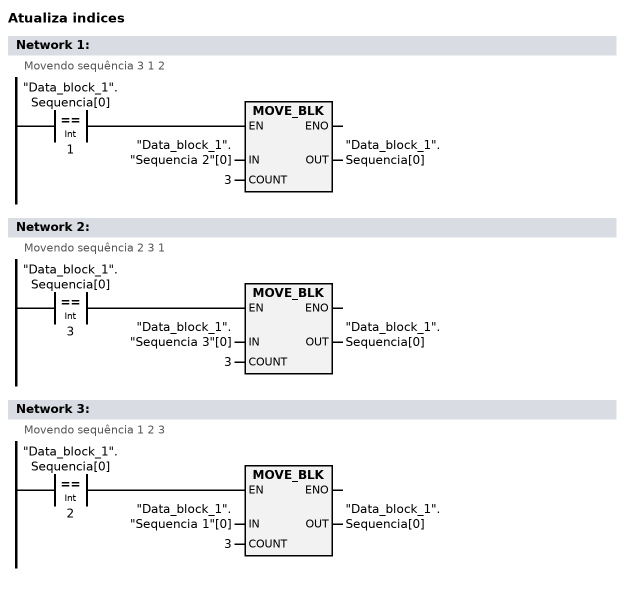
   IF "Data_block_1".Sequencia[0] = 1 THEN
       MOVE_BLK(IN := "Data_block_1"."Sequencia 2"[0], COUNT := 3, OUT => "Data_block_1".Sequencia[0]);
   END_IF;
END_REGION

REGION Network 2
   // Movendo sequência 2 3 1
   IF "Data_block_1".Sequencia[0] = 3 THEN
       MOVE_BLK(IN := "Data_block_1"."Sequencia 3"[0], COUNT := 3, OUT => "Data_block_1".Sequencia[0]);
   END_IF;
END_REGION

REGION Network 3
   // Movendo sequência 1 2 3
   IF "Data_block_1".Sequencia[0] = 2 THEN
       MOVE_BLK(IN := "Data_block_1"."Sequencia 1"[0], COUNT := 3, OUT => "Data_block_1".Sequencia[0]);
   END_IF;
END_REGION
END_FUNCTION

FUNCTION "Relaciona indices" : Void   // FC25, LAD
{ S7_Optimized_Access := 'TRUE' }
VERSION : 0.1
   VAR_INPUT
      index : Int;   // Índice da sequência de compressores
      "valor logico" : Bool;   // Valor que determina se é preciso ligar ou desligar
   END_VAR
   VAR_TEMP   // added for the SCL form of the ladder/FBD networks
      _w1 : Bool;
   END_VAR
BEGIN

REGION Network 1
   // Seta ou reseta caso Sequencia[index] == 1
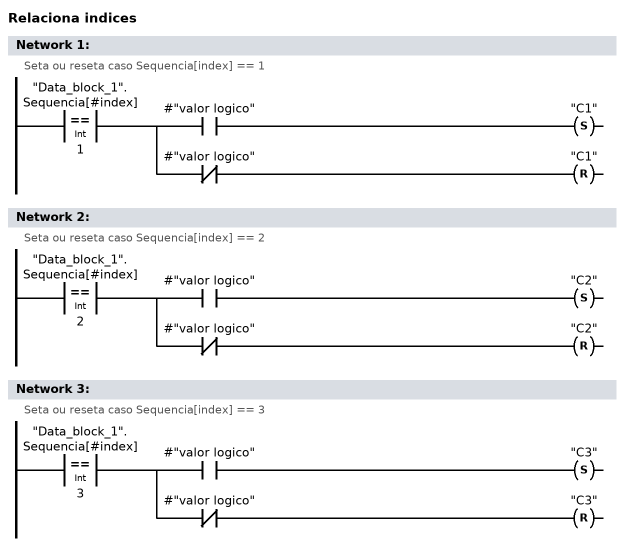
   RUNG wire#powerrail
      { S7_Templates := "SrcType := Int" } EQ_Contact(in1 := "Data_block_1".Sequencia[#index], in2 := 1)
      wire#w1
      Contact( #"valor logico" )
      S_Coil( "C1" )
   END_RUNG
   RUNG wire#w1
      I_Contact( #"valor logico" )
      R_Coil( "C1" )
   END_RUNG
   // the same network as SCL:
   #_w1 := "Data_block_1".Sequencia[#index] = 1;
   IF #_w1 AND #"valor logico" THEN "C1" := TRUE; END_IF;
   IF #_w1 AND NOT #"valor logico" THEN "C1" := FALSE; END_IF;
END_REGION

REGION Network 2
   // Seta ou reseta caso Sequencia[index] == 2
   RUNG wire#powerrail
      { S7_Templates := "SrcType := Int" } EQ_Contact(in1 := "Data_block_1".Sequencia[#index], in2 := 2)
      wire#w1
      Contact( #"valor logico" )
      S_Coil( "C2" )
   END_RUNG
   RUNG wire#w1
      I_Contact( #"valor logico" )
      R_Coil( "C2" )
   END_RUNG
   // the same network as SCL:
   #_w1 := "Data_block_1".Sequencia[#index] = 2;
   IF #_w1 AND #"valor logico" THEN "C2" := TRUE; END_IF;
   IF #_w1 AND NOT #"valor logico" THEN "C2" := FALSE; END_IF;
END_REGION

REGION Network 3
   // Seta ou reseta caso Sequencia[index] == 3
   RUNG wire#powerrail
      { S7_Templates := "SrcType := Int" } EQ_Contact(in1 := "Data_block_1".Sequencia[#index], in2 := 3)
      wire#w1
      Contact( #"valor logico" )
      S_Coil( "C3" )
   END_RUNG
   RUNG wire#w1
      I_Contact( #"valor logico" )
      R_Coil( "C3" )
   END_RUNG
   // the same network as SCL:
   #_w1 := "Data_block_1".Sequencia[#index] = 3;
   IF #_w1 AND #"valor logico" THEN "C3" := TRUE; END_IF;
   IF #_w1 AND NOT #"valor logico" THEN "C3" := FALSE; END_IF;
END_REGION
END_FUNCTION

FUNCTION "M1 - Operacao finalizada" : Void   // FC26, LAD
{ S7_Optimized_Access := 'TRUE' }
VERSION : 0.1
   VAR_TEMP   // added for the SCL form of the ladder/FBD networks
      _w1 : Bool;
   END_VAR
BEGIN

REGION Network 1
   // MODO AUTOMÁTICO [M1] - Operação finalizada
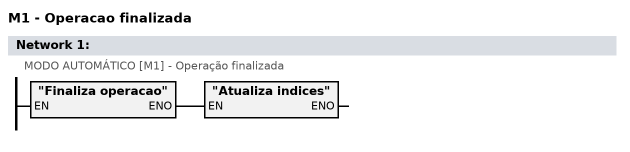
   RUNG wire#powerrail
      "Finaliza operacao"()
      "Atualiza indices"()
   END_RUNG
   // the same network as SCL:
   "Finaliza operacao"(ENO => #_w1);
   IF #_w1 THEN "Atualiza indices"(); END_IF;
END_REGION
END_FUNCTION

FUNCTION "Monitora pressao" : Void   // FC27, LAD
{ S7_Optimized_Access := 'TRUE' }
VERSION : 0.1
   VAR_OUTPUT
      Crescente : Bool;   // Pressão crescente ou decrescente
   END_VAR
   VAR_TEMP
      Pressao : Real;   // Pressao obtida
      "Positivo 1" : Bool;   // Output da função Calcula derivada
      "Positivo 2" : Bool;   // Output da função Calcula média móvel
   END_VAR
   VAR_TEMP   // added for the SCL form of the ladder/FBD networks
      _w1 : Bool;
      _w2 : Bool;
   END_VAR
BEGIN

REGION Network 1
   // Lendo pressão
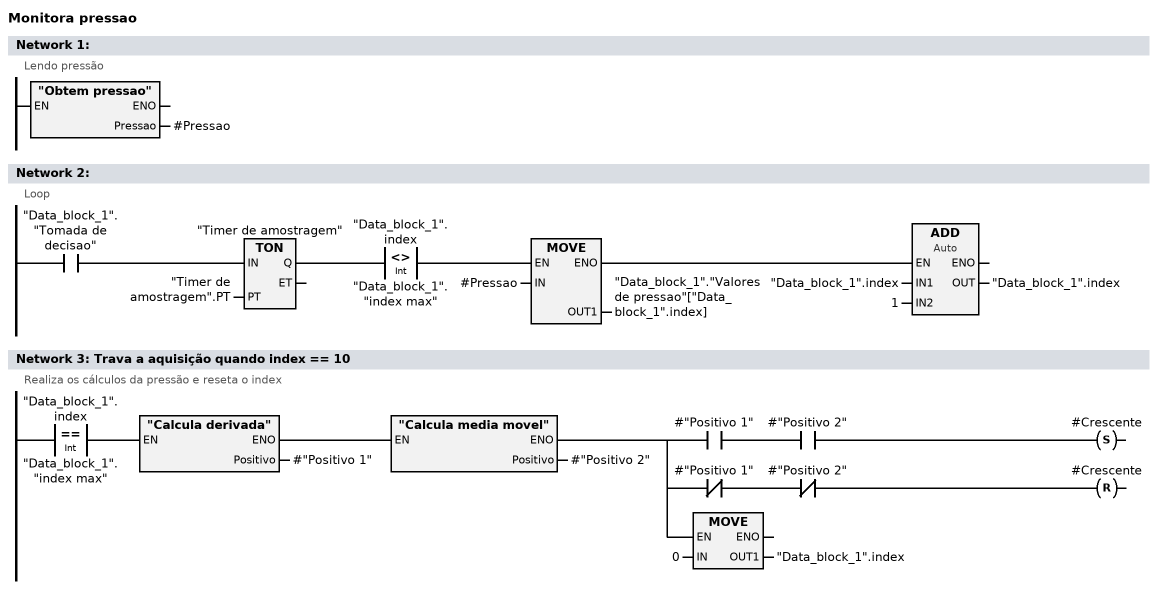
   RUNG wire#powerrail
      "Obtem pressao"(Pressao => #Pressao)
   END_RUNG
   // the same network as SCL:
   "Obtem pressao"(Pressao => #Pressao);
END_REGION

REGION Network 2
   // Loop
   "Timer de amostragem".TON(IN := "Data_block_1"."Tomada de decisao", PT := "Timer de amostragem".PT);
   #_w1 := "Timer de amostragem".Q AND ("Data_block_1".index <> "Data_block_1"."index max");
   IF #_w1 THEN
       "Data_block_1"."Valores de pressao"["Data_block_1".index] := #Pressao;
       "Data_block_1".index := "Data_block_1".index + 1;
   END_IF;
END_REGION

REGION Network 3: Trava a aquisição quando index == 10
   // Realiza os cálculos da pressão e reseta o index
   RUNG wire#powerrail
      { S7_Templates := "SrcType := Int" } EQ_Contact(in1 := "Data_block_1".index, in2 := "Data_block_1"."index max")
      "Calcula derivada"(Positivo => #"Positivo 1")
      "Calcula media movel"(Positivo => #"Positivo 2")
      wire#w1
      Contact( #"Positivo 1" )
      Contact( #"Positivo 2" )
      S_Coil( #Crescente )
   END_RUNG
   RUNG wire#w1
      I_Contact( #"Positivo 1" )
      I_Contact( #"Positivo 2" )
      R_Coil( #Crescente )
   END_RUNG
   RUNG wire#w1
      Move(in := 0, out1 => "Data_block_1".index)
   END_RUNG
   // the same network as SCL:
   "Calcula derivada"(EN := "Data_block_1".index = "Data_block_1"."index max",
                      Positivo => #"Positivo 1",
                      ENO => #_w1);
   "Calcula media movel"(EN := #_w1, Positivo => #"Positivo 2", ENO => #_w2);
   IF #_w2 AND #"Positivo 1" AND #"Positivo 2" THEN #Crescente := TRUE; END_IF;
   IF #_w2 AND NOT #"Positivo 1" AND NOT #"Positivo 2" THEN #Crescente := FALSE; END_IF;
   IF #_w2 THEN "Data_block_1".index := 0; END_IF;
END_REGION
END_FUNCTION

FUNCTION "Calcula media movel" : Void   // FC28, LAD
{ S7_Optimized_Access := 'TRUE' }
VERSION : 0.1
   VAR_OUTPUT
      Positivo : Bool;
   END_VAR
   VAR_TEMP
      "Soma 5" : Real;
      "Soma 10" : Real;
      "index 5" : Int;
      "index 10" : Int;
      "Media 5" : Real;
      "Media 10" : Real;
   END_VAR
BEGIN

REGION Network 1 (SCL)
   // Calcula média dos 5 primeiros valores
   #"Soma 5" := 0.0;
   #"Media 5" := 0.0;

   FOR #"index 5" := 0 TO 4 DO
       // Statement section FOR
       #"Soma 5" += "Data_block_1"."Valores de pressao"[#"index 5"];
   END_FOR;

   #"Media 5" := #"Soma 5" / (#"index 5" + 1);
END_REGION

REGION Network 2 (SCL)
   // Calcula média de todos os valores
   #"Soma 10" := 0.0;
   #"Media 10" := 0.0;

   FOR #"index 10" := 0 TO 9 DO
       // Statement section FOR
       #"Soma 10" += "Data_block_1"."Valores de pressao"[#"index 10"];
   END_FOR;

   #"Media 10" := #"Soma 10" / (#"index 10" + 1);
END_REGION

REGION Network 3
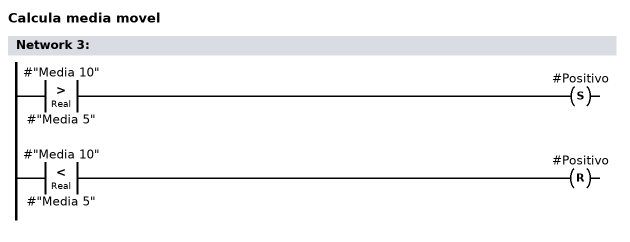
   RUNG wire#powerrail
      { S7_Templates := "SrcType := Real" } GT_Contact(in1 := #"Media 10", in2 := #"Media 5")
      S_Coil( #Positivo )
   END_RUNG
   RUNG wire#powerrail
      { S7_Templates := "SrcType := Real" } LT_Contact(in1 := #"Media 10", in2 := #"Media 5")
      R_Coil( #Positivo )
   END_RUNG
   // the same network as SCL:
   IF #"Media 10" > #"Media 5" THEN #Positivo := TRUE; END_IF;
   IF #"Media 10" < #"Media 5" THEN #Positivo := FALSE; END_IF;
END_REGION
END_FUNCTION

FUNCTION "Calcula derivada" : Void   // FC29, LAD
{ S7_Optimized_Access := 'TRUE' }
VERSION : 0.1
   VAR_OUTPUT
      Positivo : Bool;   // Indica se dP/dt > 0
   END_VAR
   VAR_TEMP
      Derivada : Real;
   END_VAR
BEGIN

REGION Network 1
   // Calcula a derivada
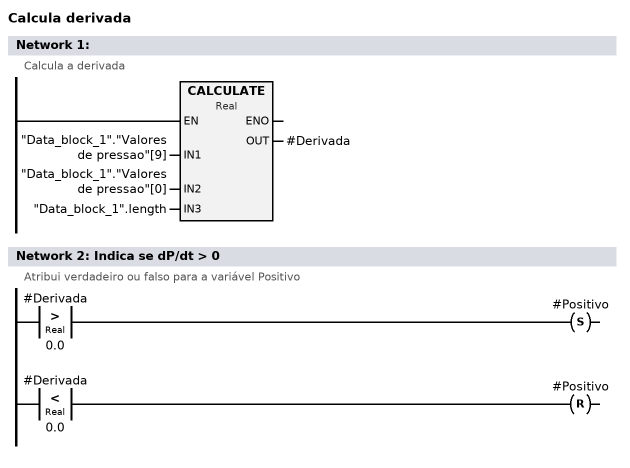
   RUNG wire#powerrail
      { S7_Templates := "SrcType := Real"; S7_Expression := "(IN1 - IN2) / IN3" } Calculate(in1 := "Data_block_1"."Valores de pressao"[9], in2 := "Data_block_1"."Valores de pressao"[0], in3 := "Data_block_1".length, out => #Derivada)
   END_RUNG
   // the same network as SCL:
   #Derivada := ("Data_block_1"."Valores de pressao"[9] - "Data_block_1"."Valores de pressao"[0]) / "Data_block_1".length;
END_REGION

REGION Network 2: Indica se dP/dt > 0
   // Atribui verdadeiro ou falso para a variável Positivo
   RUNG wire#powerrail
      { S7_Templates := "SrcType := Real" } GT_Contact(in1 := #Derivada, in2 := 0.0)
      S_Coil( #Positivo )
   END_RUNG
   RUNG wire#powerrail
      { S7_Templates := "SrcType := Real" } LT_Contact(in1 := #Derivada, in2 := 0.0)
      R_Coil( #Positivo )
   END_RUNG
   // the same network as SCL:
   IF #Derivada > 0.0 THEN #Positivo := TRUE; END_IF;
   IF #Derivada < 0.0 THEN #Positivo := FALSE; END_IF;
END_REGION
END_FUNCTION

FUNCTION "M1 - Operacao iniciada" : Void   // FC30, LAD
{ S7_Optimized_Access := 'TRUE' }
VERSION : 0.1
   VAR_TEMP
      Crescente : Bool;   // Output da função Monitora pressão
      P : Real;   // Pressão no interior do tanque separador
   END_VAR
   VAR_TEMP   // added for the SCL form of the ladder/FBD networks
      _w1 : Bool;
   END_VAR
BEGIN

REGION Network 1
   // MODO AUTOMÁTICO [M1] - Operação iniciada
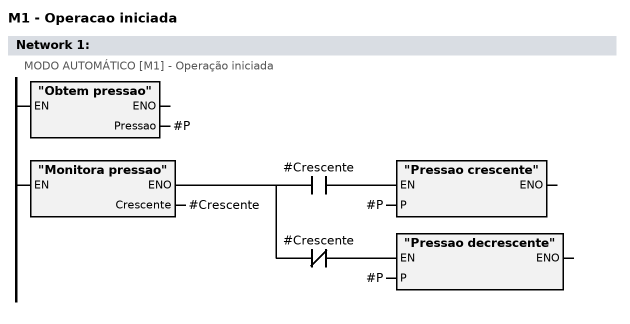
   RUNG wire#powerrail
      "Obtem pressao"(Pressao => #P)
   END_RUNG
   RUNG wire#powerrail
      "Monitora pressao"(Crescente => #Crescente)
      wire#w1
      Contact( #Crescente )
      "Pressao crescente"(P := #P)
   END_RUNG
   RUNG wire#w1
      I_Contact( #Crescente )
      "Pressao decrescente"(P := #P)
   END_RUNG
   // the same network as SCL:
   "Obtem pressao"(Pressao => #P);
   "Monitora pressao"(Crescente => #Crescente, ENO => #_w1);
   IF #_w1 AND #Crescente THEN "Pressao crescente"(P := #P); END_IF;
   IF #_w1 AND NOT #Crescente THEN "Pressao decrescente"(P := #P); END_IF;
END_REGION
END_FUNCTION

FUNCTION "Obtem pressao de saida" : Void   // FC31, LAD
{ S7_Optimized_Access := 'TRUE' }
VERSION : 0.1
   VAR_OUTPUT
      "Pressao saida" : Real;   // Pressão na saída do conjunto de compressores
   END_VAR
   VAR_TEMP
      "Pressao normalizada" : Real;   // Pressão de saída normalizada
   END_VAR
BEGIN

REGION Network 1
   // Normalização do valor de pressão lido do transmissor
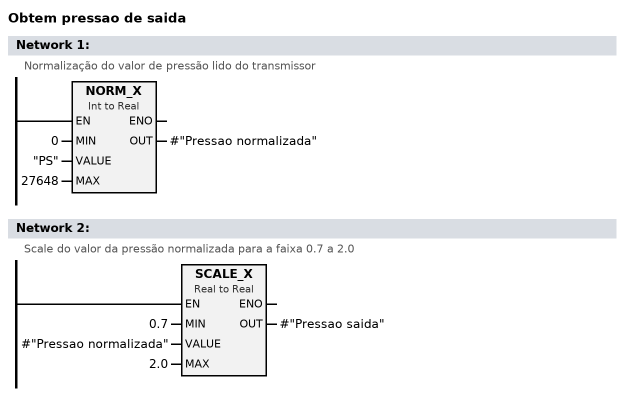
   RUNG wire#powerrail
      { S7_Templates := "[SrcType := Int, DestType := Real]" } Normalize(min := 0, value := "PS", max := 27648, out => #"Pressao normalizada")
   END_RUNG
   // the same network as SCL:
   #"Pressao normalizada" := NORM_X(MIN := 0, VALUE := "PS", MAX := 27648);
END_REGION

REGION Network 2
   // Scale do valor da pressão normalizada para a faixa 0.7 a 2.0
   RUNG wire#powerrail
      { S7_Templates := "[SrcType := Real, DestType := Real]" } Scale(min := 0.7, value := #"Pressao normalizada", max := 2.0, out => #"Pressao saida")
   END_RUNG
   // the same network as SCL:
   #"Pressao saida" := SCALE_X(MIN := 0.7, VALUE := #"Pressao normalizada", MAX := 2.0);
END_REGION
END_FUNCTION

FUNCTION "Obtem pressao - M3" : Void   // FC32, LAD
{ S7_Optimized_Access := 'TRUE' }
VERSION : 0.1
   VAR_OUTPUT
      "Pressao abastecimento" : Real;   // Pressão no nó estendido
   END_VAR
   VAR_TEMP
      "Pressao normalizada" : Real;   // Pressão normalizada
   END_VAR
BEGIN

REGION Network 1
   // Normalização do valor de pressão lido do transmissor
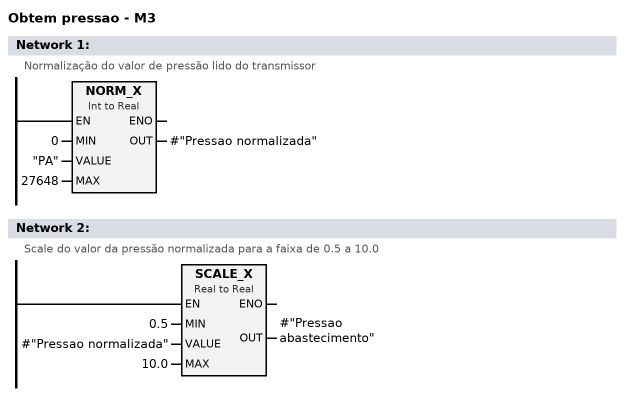
   RUNG wire#powerrail
      { S7_Templates := "[SrcType := Int, DestType := Real]" } Normalize(min := 0, value := "PA", max := 27648, out => #"Pressao normalizada")
   END_RUNG
   // the same network as SCL:
   #"Pressao normalizada" := NORM_X(MIN := 0, VALUE := "PA", MAX := 27648);
END_REGION

REGION Network 2
   // Scale do valor da pressão normalizada para a faixa de 0.5 a 10.0
   RUNG wire#powerrail
      { S7_Templates := "[SrcType := Real, DestType := Real]" } Scale(min := 0.5, value := #"Pressao normalizada", max := 10.0, out => #"Pressao abastecimento")
   END_RUNG
   // the same network as SCL:
   #"Pressao abastecimento" := SCALE_X(MIN := 0.5, VALUE := #"Pressao normalizada", MAX := 10.0);
END_REGION
END_FUNCTION

FUNCTION "Calcula media - M3" : Void   // FC33, LAD
{ S7_Optimized_Access := 'TRUE' }
VERSION : 0.1
   VAR_OUTPUT
      Media : Real;   // Média dos valores de pressão
   END_VAR
   VAR_TEMP
      index : Int;
      soma : Real;
   END_VAR
BEGIN

REGION Network 1 (SCL)
   // Calculando a média dos valores de pressão
   #index := 0;
   #soma := 0.0;
   #Media := 0.0;

   FOR #index := 0 TO "Data_block_1"."length - M3" - 1 DO
       // Statement section FOR
       #soma += "Data_block_1"."Valores de pressao - M3"[#index];
   END_FOR;

   #Media := #soma / "Data_block_1"."length - M3";
END_REGION
END_FUNCTION

FUNCTION "M3 - Operacao iniciada" : Void   // FC34, LAD
{ S7_Optimized_Access := 'TRUE' }
VERSION : 0.1
// MODO ABASTECIMENTO [M3] - Operação iniciada
   VAR_TEMP
      Media : Real;   // Média dos valores de pressão
      "Threshold de Peq" : Real;   // (1 - gamma)*Peq
   END_VAR
   VAR_TEMP   // added for the SCL form of the ladder/FBD networks
      _w1 : Bool;
   END_VAR
BEGIN

REGION Network 1
   // Acionando válvulas da linha direta
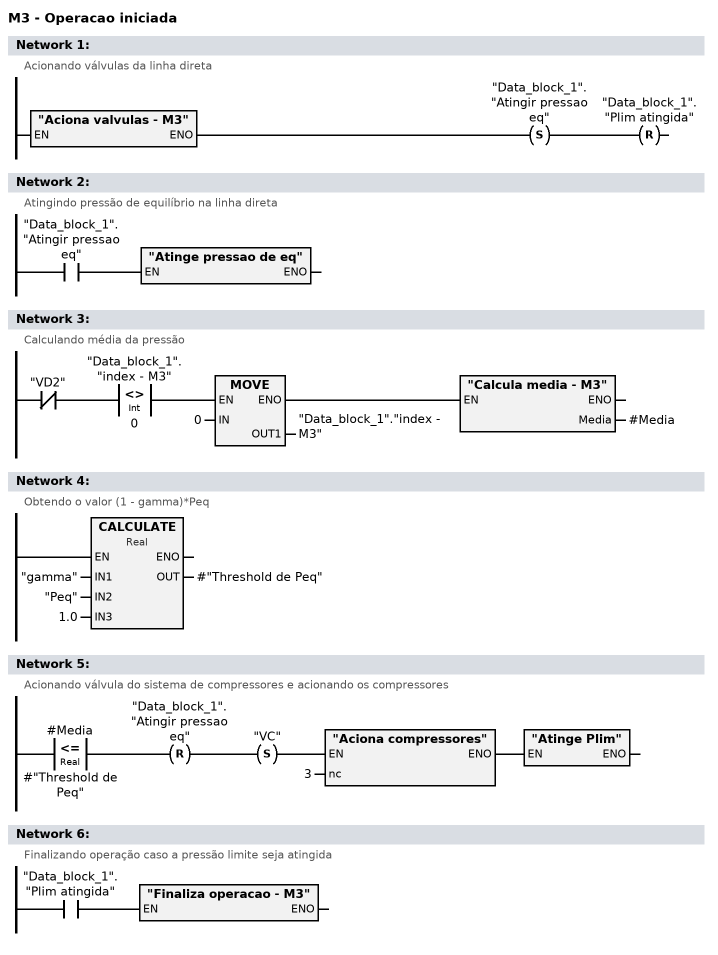
   RUNG wire#powerrail
      "Aciona valvulas - M3"()
      S_Coil( "Data_block_1"."Atingir pressao eq" )
      R_Coil( "Data_block_1"."Plim atingida" )
   END_RUNG
   // the same network as SCL:
   "Aciona valvulas - M3"(ENO => #_w1);
   IF #_w1 THEN
       "Data_block_1"."Atingir pressao eq" := TRUE;
       "Data_block_1"."Plim atingida" := FALSE;
   END_IF;
END_REGION

REGION Network 2
   // Atingindo pressão de equilíbrio na linha direta
   RUNG wire#powerrail
      Contact( "Data_block_1"."Atingir pressao eq" )
      "Atinge pressao de eq"()
   END_RUNG
   // the same network as SCL:
   IF "Data_block_1"."Atingir pressao eq" THEN "Atinge pressao de eq"(); END_IF;
END_REGION

REGION Network 3
   // Calculando média da pressão
   RUNG wire#powerrail
      I_Contact( "VD2" )
      { S7_Templates := "SrcType := Int" } NE_Contact(in1 := "Data_block_1"."index - M3", in2 := 0)
      Move(in := 0, out1 => "Data_block_1"."index - M3")
      "Calcula media - M3"(Media => #Media)
   END_RUNG
   // the same network as SCL:
   #_w1 := NOT "VD2" AND ("Data_block_1"."index - M3" <> 0);
   IF #_w1 THEN
       "Data_block_1"."index - M3" := 0;
       "Calcula media - M3"(Media => #Media);
   END_IF;
END_REGION

REGION Network 4
   // Obtendo o valor (1 - gamma)*Peq
   RUNG wire#powerrail
      { S7_Templates := "SrcType := Real"; S7_Expression := "(IN3 - IN1) * IN2" } Calculate(in1 := "gamma", in2 := "Peq", in3 := 1.0, out => #"Threshold de Peq")
   END_RUNG
   // the same network as SCL:
   #"Threshold de Peq" := (1.0 - "gamma") * "Peq";
END_REGION

REGION Network 5
   // Acionando válvula do sistema de compressores e acionando os compressores
   RUNG wire#powerrail
      { S7_Templates := "SrcType := Real" } LE_Contact(in1 := #Media, in2 := #"Threshold de Peq")
      R_Coil( "Data_block_1"."Atingir pressao eq" )
      S_Coil( "VC" )
      "Aciona compressores"(nc := 3)
      "Atinge Plim"()
   END_RUNG
   // the same network as SCL:
   IF #Media <= #"Threshold de Peq" THEN
       "Data_block_1"."Atingir pressao eq" := FALSE;
       "VC" := TRUE;
   END_IF;
   "Aciona compressores"(EN := #Media <= #"Threshold de Peq", nc := 3, ENO => #_w1);
   IF #_w1 THEN "Atinge Plim"(); END_IF;
END_REGION

REGION Network 6
   // Finalizando operação caso a pressão limite seja atingida
   RUNG wire#powerrail
      Contact( "Data_block_1"."Plim atingida" )
      "Finaliza operacao - M3"()
   END_RUNG
   // the same network as SCL:
   IF "Data_block_1"."Plim atingida" THEN "Finaliza operacao - M3"(); END_IF;
END_REGION
END_FUNCTION

FUNCTION "Atinge Plim" : Void   // FC35, LAD
{ S7_Optimized_Access := 'TRUE' }
VERSION : 0.1
   VAR_TEMP
      "Pressao abastecimento" : Real;
   END_VAR
BEGIN

REGION Network 1
   // Obtém pressão de abastecimento
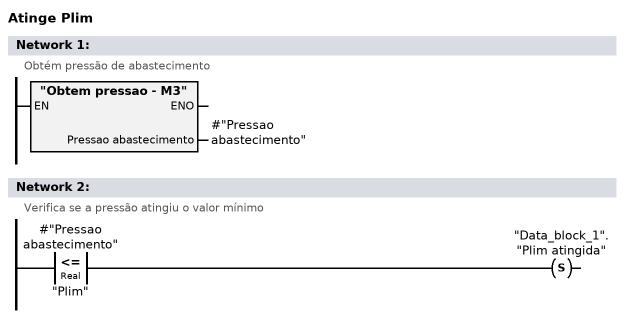
   RUNG wire#powerrail
      "Obtem pressao - M3"("Pressao abastecimento" => #"Pressao abastecimento")
   END_RUNG
   // the same network as SCL:
   "Obtem pressao - M3"("Pressao abastecimento" => #"Pressao abastecimento");
END_REGION

REGION Network 2
   // Verifica se a pressão atingiu o valor mínimo
   RUNG wire#powerrail
      { S7_Templates := "SrcType := Real" } LE_Contact(in1 := #"Pressao abastecimento", in2 := "Plim")
      S_Coil( "Data_block_1"."Plim atingida" )
   END_RUNG
   // the same network as SCL:
   IF #"Pressao abastecimento" <= "Plim" THEN "Data_block_1"."Plim atingida" := TRUE; END_IF;
END_REGION
END_FUNCTION

FUNCTION "Desliga valvulas - M3" : Void   // FC36, LAD
{ S7_Optimized_Access := 'TRUE' }
VERSION : 0.1
BEGIN

REGION Network 1
   // Desliga as válvulas da linha direta
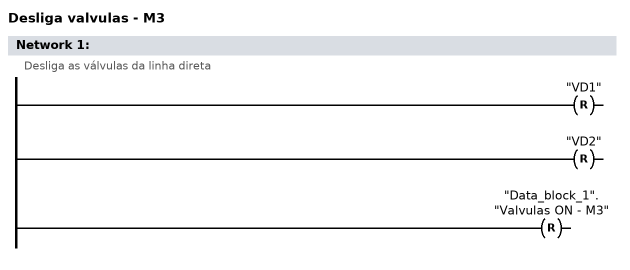
   RUNG wire#powerrail
      R_Coil( "VD1" )
   END_RUNG
   RUNG wire#powerrail
      R_Coil( "VD2" )
   END_RUNG
   RUNG wire#powerrail
      R_Coil( "Data_block_1"."Valvulas ON - M3" )
   END_RUNG
   // the same network as SCL:
   "VD1" := FALSE;
   "VD2" := FALSE;
   "Data_block_1"."Valvulas ON - M3" := FALSE;
END_REGION
END_FUNCTION

FUNCTION "Verifica valvulas 3" : Void   // FC37, LAD
{ S7_Optimized_Access := 'TRUE' }
VERSION : 0.1
BEGIN

REGION Network 1
   // Desliga as válvulas da linha direta caso estejam ligadas
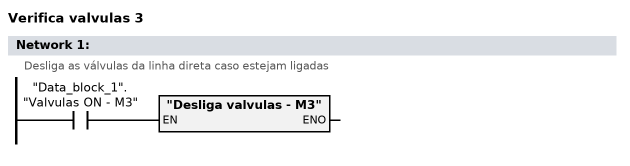
   RUNG wire#powerrail
      Contact( "Data_block_1"."Valvulas ON - M3" )
      "Desliga valvulas - M3"()
   END_RUNG
   // the same network as SCL:
   IF "Data_block_1"."Valvulas ON - M3" THEN "Desliga valvulas - M3"(); END_IF;
END_REGION
END_FUNCTION

FUNCTION "Finaliza operacao - M3" : Void   // FC38, LAD
{ S7_Optimized_Access := 'TRUE' }
VERSION : 0.1
   VAR_TEMP   // added for the SCL form of the ladder/FBD networks
      _w1 : Bool;
      _w2 : Bool;
   END_VAR
BEGIN

REGION Network 1
   // Finalizando operação - M3
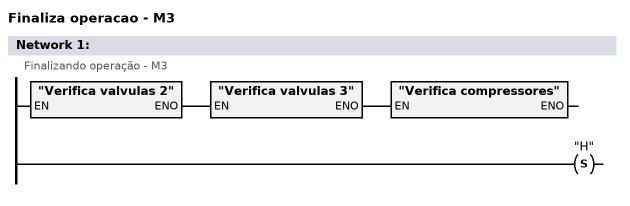
   RUNG wire#powerrail
      "Verifica valvulas 2"()
      "Verifica valvulas 3"()
      "Verifica compressores"()
   END_RUNG
   RUNG wire#powerrail
      S_Coil( "H" )
   END_RUNG
   // the same network as SCL:
   "Verifica valvulas 2"(ENO => #_w1);
   "Verifica valvulas 3"(EN := #_w1, ENO => #_w2);
   IF #_w2 THEN "Verifica compressores"(); END_IF;
   "H" := TRUE;
END_REGION
END_FUNCTION

FUNCTION "M3 - Operacao finalizada" : Void   // FC39, LAD
{ S7_Optimized_Access := 'TRUE' }
VERSION : 0.1
BEGIN

REGION Network 1
   // MODO ABASTECIMENTO [M3] - Operação finalizada
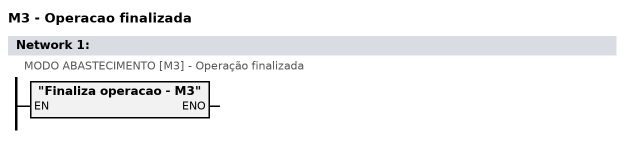
   RUNG wire#powerrail
      "Finaliza operacao - M3"()
   END_RUNG
   // the same network as SCL:
   "Finaliza operacao - M3"();
END_REGION
END_FUNCTION

ORGANIZATION_BLOCK "Main"   // OB1, LAD, ProgramCycle
TITLE = "Main Program Sweep (Cycle)"
{ S7_Optimized_Access := 'TRUE' }
VERSION : 0.1
   VAR_INPUT
      Initial_Call : Bool;   // Initial call of this OB
      Remanence : Bool;   // =True, if remanent data are available
   END_VAR
BEGIN

REGION Network 1
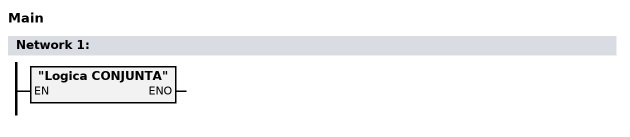
   RUNG wire#powerrail
      "Logica CONJUNTA"()
   END_RUNG
   // the same network as SCL:
   "Logica CONJUNTA"();
END_REGION
END_ORGANIZATION_BLOCK